Fanuc TP program (LS listing): ESB_TEST_F9.LS

/PROG  ESB_TEST_F9
/ATTR
OWNER		= MNEDITOR;
COMMENT		= "TEST PROGRAM";
PROG_SIZE	= 3071;
CREATE		= DATE 29-01-26  TIME 08:00:00;
MODIFIED	= DATE 29-01-26  TIME 08:00:00;
FILE_NAME	= ESB_TEST_F9;
VERSION		= 0;
LINE_COUNT	= 100;
MEMORY_SIZE	= 3515;
PROTECT		= READ_WRITE;
TCD:  STACK_SIZE	= 0,
      TASK_PRIORITY	= 50,
      TIME_SLICE	= 0,
      BUSY_LAMP_OFF	= 0,
      ABORT_REQUEST	= 0,
      PAUSE_REQUEST	= 0;
DEFAULT_GROUP	= 1,*,*,*,*;
CONTROL_CODE	= 00000000 00000000;
/APPL

AUTO_SINGULARITY_HEADER;
  ENABLE_SINGULARITY_AVOIDANCE   : TRUE;
/MN
   1:  MESSAGE[This is a test !] ;
   2:  UFRAME_NUM = 0 ;
   3:  UTOOL_NUM  = 1 ;
   4:  J PR[1] 50% FINE ;
   5:  WAIT  1.0(sec) ;
   6:  PR[300] =LPOS  ;
   7:  PR[300,3] = PR[300,3] + 500 ;
   8:  ! PR[300,2] = 0 ;
   9:  ! PR[300,3] = 0 ;
 10:  UFRAME_NUM = 12 ;
 11:  UTOOL_NUM = 1;
 12:   L  PR[300] 200mm/sec FINE ;
/POS
/END
